TYPE ST_Panel :
STRUCT
	Name				: STRING(255);
	InstanzName			: STRING(255);
	Button				: BOOL;
	InsertCoin			: BOOL;
	TakeProduct			: BOOL;
	TakeCoin			: BOOL;
	State				: STRING;
	NumberOfProducts	: UINT;
END_STRUCT
END_TYPE

(* stored: Version 1.1.0.1, ProductVersion 3.1.4024.9
   DUT ST_Panel: Id {41dd766d-599b-4936-8647-4842b7cb5f29} *)
